Universal Robots PolyScope program: NICOL.urp

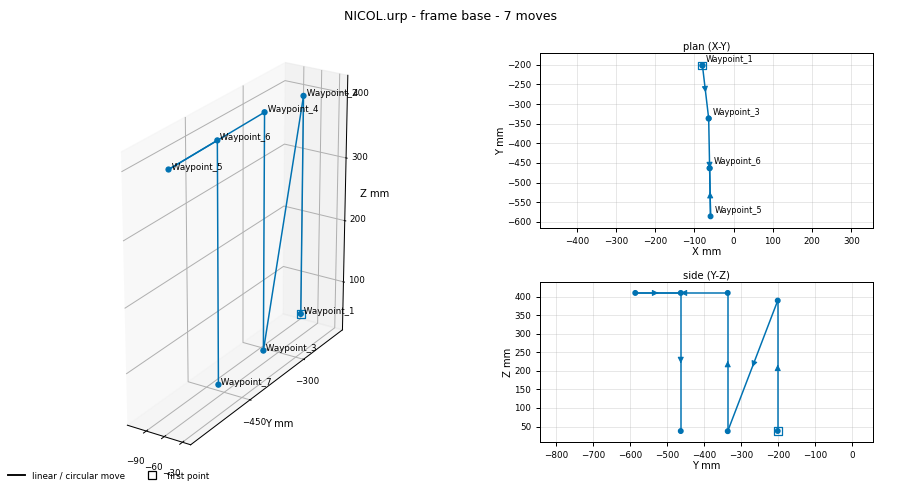
[picture p0: tool path of NICOL.urp in frame base, 7 of 7 moves have a stored position in this frame; points joined in program order, loops and branches not executed]
Program NICOL (installation=default directory=/ursim/programs createdIn=3.15.8.106339 lastSavedIn=3.15.8.106339 robotSerialNumber=2018359999)
Calibrated DH parameters: a=[0, -0.425, -0.39225, 0, 0, 0]; d=[0.089159, 0, 0, 0.10915, 0.09465, 0.0823]; alpha=[1.570796, 0, 0, 1.570796, -1.570796, 0]; deltaTheta=[0, 0, 0, 0, 0, 0]
Robot Program (runOnlyOnce=false)
  Popup Message (haltProgram=false message=Se dibujara la letra N y T inputType=Text)
  MoveL speed 250 mm/s, acceleration 1200 mm/s^2 (useActiveTCP=true) feature=Base
    Waypoint Waypoint_1: TCP in base x=-79.473 y=-201.665 z=37.972 mm, rx=0.0064 ry=-2.1379 rz=-2.236 rad; joints [-83.288, -108.091, -140.171, -114.345, 94.636, 1.52] deg
    Waypoint Waypoint_2: TCP in base x=-79.473 y=-201.665 z=389.97 mm, rx=0.0064 ry=-2.1379 rz=-2.236 rad; joints [-83.288, -74.356, -108.22, -180.032, 94.636, 1.52] deg
    Waypoint Waypoint_3: TCP in base x=-63.588 y=-336.641 z=37.35 mm, rx=-0.097 ry=-0.5173 rz=-2.9675 rad; joints [-83.288, -139.517, -112.624, -178.305, 94.636, 1.52] deg
    Waypoint Waypoint_4: TCP in base x=-63.588 y=-336.641 z=410.549 mm, rx=-0.097 ry=-0.5173 rz=-2.9675 rad; joints [-83.288, -100.564, -100.665, -229.218, 94.636, 1.52] deg
    Waypoint Waypoint_5: TCP in base x=-58.82 y=-586.194 z=410.549 mm, rx=-0.097 ry=-0.5173 rz=-2.9675 rad; joints [-85.601, -135.863, -47.05, -247.371, 93.858, 3.704] deg
    Waypoint Waypoint_6: TCP in base x=-61.166 y=-463.421 z=410.549 mm, rx=-0.097 ry=-0.5173 rz=-2.9675 rad; joints [-84.763, -117.153, -77.953, -235.233, 94.141, 2.914] deg
    Waypoint Waypoint_7: TCP in base x=-61.166 y=-463.421 z=37.75 mm, rx=-0.097 ry=-0.5173 rz=-2.9675 rad; joints [-84.763, -147.119, -89.514, -193.707, 94.141, 2.914] deg
